FUNCTION GetXSide : LREAL
VAR_INPUT
	xPos : LREAL;
END_VAR
VAR
END_VAR

GetXSide := GVL_RobotArmConstants.DISTANCE_TO_PICKUP_AREA + xPos;

END_FUNCTION

(* stored: Version 1.1.0.1, ProductVersion 3.1.4024.12
   POU GetXSide: Id {e81490c4-9833-4755-8734-64c7883bf73b}, SpecialFunc None *)
